(* Visualisation VIS_SET
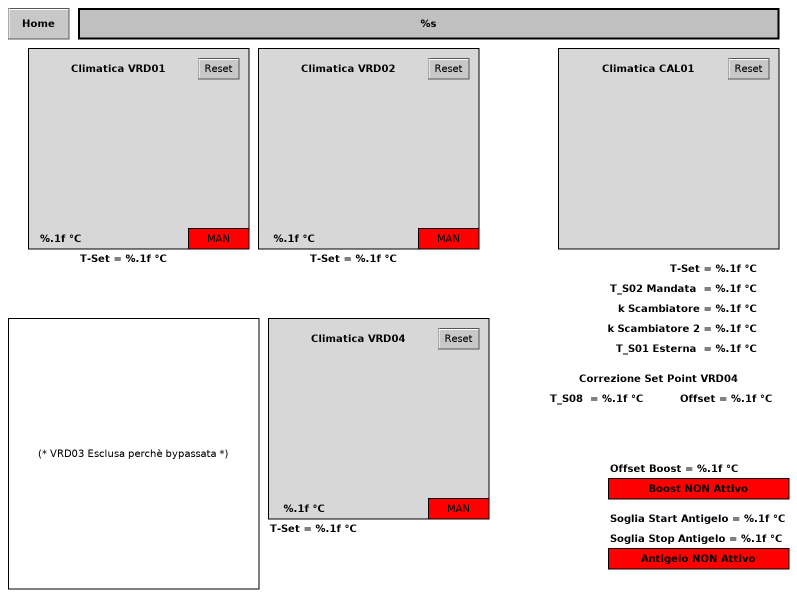
rectangle at (40,60)-(201,81): text "Climatica VRD01"
button at (200,60)-(241,81): text "Reset"; taps .VRD01.CLIM.InitOK
button at (10,10)-(71,41): text "Home"; opens PLC_VISU
rectangle at (80,250)-(221,271): text "T-Set = %.1f °C"; shows INT_TO_REAL(.VRD01.SetPoint)/10
rectangle at (270,60)-(431,81): text "Climatica VRD02"
button at (430,60)-(471,81): text "Reset"; taps .VRD02.CLIM.InitOK; runs INTERN ASSIGN VRD02_Clima.InitOK:=(FALSE)
rectangle at (310,250)-(451,271): text "T-Set = %.1f °C"; shows INT_TO_REAL(.VRD02.SetPoint)/10
rectangle at (40,230)-(91,251): text "%.1f °C"; shows INT_TO_REAL(.TPV04.IN)/10
rectangle at (270,230)-(321,251): text "%.1f °C"; shows INT_TO_REAL(.TPV05.IN)/10
rectangle at (570,60)-(731,81): text "Climatica CAL01"
button at (730,60)-(771,81): text "Reset"; taps .VRD02.CLIM.InitOK; runs INTERN ASSIGN VRD02_Clima.InitOK:=(FALSE)
rectangle at (620,260)-(761,281): text "T-Set = %.1f °C"; shows INT_TO_REAL(.CAL01.SetPoint)/10
rectangle at (80,10)-(781,41): text "%s"; shows .Plant_NAME
rectangle at (40,330)-(201,351): text "Climatica VRD03"
button at (200,330)-(241,351): text "Reset"; taps .VRD03.CLIM.InitOK; runs INTERN ASSIGN VRD02_Clima.InitOK:=(FALSE)
rectangle at (70,520)-(211,541): text "T-Set = %.1f °C"; shows INT_TO_REAL(.VRD03.Ctrl_SetPoint)/10
rectangle at (40,500)-(91,521): text "%.1f °C"; shows INT_TO_REAL(.TPV06.IN)/10
rectangle at (600,300)-(761,321): text "k Scambiatore = %.1f °C"; shows INT_TO_REAL(.OffsetSetPointManuale/10)
rectangle at (280,330)-(441,351): text "Climatica VRD04"
button at (440,330)-(481,351): text "Reset"; taps .VRD04.CLIM.InitOK; runs INTERN ASSIGN VRD02_Clima.InitOK:=(FALSE)
rectangle at (270,520)-(391,541): text "T-Set = %.1f °C"; shows INT_TO_REAL(.VRD04.SetPoint)/10
rectangle at (280,500)-(331,521): text "%.1f °C"; shows INT_TO_REAL(.TPV09.AVG)/10
rectangle at (190,230)-(251,251): text "MAN"; invisible if NOT .VRD01.ComandoManuale
rectangle at (420,230)-(481,251): text "MAN"; invisible if NOT .VRD02.ComandoManuale
rectangle at (190,500)-(251,521): text "MAN"; invisible if NOT .VRD03.ComandoManuale
rectangle at (430,500)-(491,521): text "MAN"; invisible if NOT .VRD04.ComandoManuale
rectangle at (600,320)-(761,341): text "k Scambiatore 2 = %.1f °C"; shows INT_TO_REAL(.OffsetSetPointManuale2/10)
rectangle at (610,460)-(791,481): text "Offset Boost = %.1f °C"; shows INT_TO_REAL(.RifOffsetBoost/10)
rectangle at (610,480)-(791,501): text "Boost Attivo"; invisible if NOT .BitAbilitaBoost
rectangle at (610,480)-(791,501): text "Boost NON Attivo"; invisible if .BitAbilitaBoost
rectangle at (10,320)-(261,591): text "( * VRD03 Esclusa perchè bypassata * )"
rectangle at (610,510)-(791,531): text "Soglia Start Antigelo = %.1f °C"; shows INT_TO_REAL((.SogliaMinStartAntigelo)/10)
rectangle at (610,550)-(791,571): text "Antigleo Attivo"; invisible if NOT .PLC_PRG.StartCAL_Antigelo.Q1
rectangle at (610,550)-(791,571): text "Antigelo NON Attivo"; invisible if .PLC_PRG.StartCAL_Antigelo.Q1
rectangle at (610,530)-(791,551): text "Soglia Stop Antigelo = %.1f °C"; shows INT_TO_REAL((.SogliaMinStopAntigelo)/10)
rectangle at (590,340)-(761,361): text "T_S01 Esterna  = %.1f °C"; shows INT_TO_REAL(.TPV01.IN)/10
rectangle at (600,280)-(761,301): text "T_S02 Mandata  = %.1f °C"; shows INT_TO_REAL(.TPV02.AVG)/10
rectangle at (550,370)-(771,391): text "Correzione Set Point VRD04"
rectangle at (550,390)-(661,411): text "T_S08  = %.1f °C"; shows INT_TO_REAL(.TPV08.IN)/10
rectangle at (680,390)-(791,411): text "Offset = %.1f °C"; shows INT_TO_REAL(PLC_PRG.OffsetVRD04)/10
6 more shapes without text or variables
81 elements of other kinds (tables, trends, ...) not read
*)
